{attribute 'GeneratedUsingTerminal: EL6201-0000-0017'}
{attribute addProperty BoxType "EL6201-0000-0017"}
{attribute addProperty Id "Slave_10A_DI0BOOL1Slave_10A_DI1BOOL1Slave_10A_DI2BOOL1Slave_10A_DI3BOOL1Slave_10B_DI0BOOL1Slave_10B_DI1BOOL1Slave_10B_DI2BOOL1Slave_10B_DI3BOOL1"}
{attribute addProperty CRC "31874685"}
{attribute addProperty Size "8"}
TYPE Slave_10_Inputs_01E65E7D :
STRUCT
	{attribute addProperty Name "Slave_10A_DI0"}
	Slave_10A_DI0 : BOOL;
	{attribute addProperty Name "Slave_10A_DI1"}
	Slave_10A_DI1 : BOOL;
	{attribute addProperty Name "Slave_10A_DI2"}
	Slave_10A_DI2 : BOOL;
	{attribute addProperty Name "Slave_10A_DI3"}
	Slave_10A_DI3 : BOOL;
	{attribute addProperty Name "Slave_10B_DI0"}
	Slave_10B_DI0 : BOOL;
	{attribute addProperty Name "Slave_10B_DI1"}
	Slave_10B_DI1 : BOOL;
	{attribute addProperty Name "Slave_10B_DI2"}
	Slave_10B_DI2 : BOOL;
	{attribute addProperty Name "Slave_10B_DI3"}
	Slave_10B_DI3 : BOOL;
END_STRUCT
END_TYPE

(* stored: Version 1.2.0.0, ProductVersion 3.1.4024.9
   DUT Slave_10_Inputs_01E65E7D: Id {314f7450-179e-4775-95a0-e649e8ed404f} *)
